// TIA Portal V19 export
TYPE "LEXCHANGETRAY_typeNgConveyor_deliver_interface"
// stored: Access Published
   STRUCT
      init : Bool;
      handlingXyz : "LEXCHANGETRAY_typeNgConveyor_toHandlingXyzDeliver";
   END_STRUCT;
END_TYPE
